TYPE ST_TcMatSimObjectDataAreaInfo :
STRUCT
	pPlcVar: PVOID;
	pModuleProcImg: PVOID;
	nSize: UDINT;
	nDataAreaId: UDINT;
	eDataAreaType: E_TcMatSimDataAreaType;
END_STRUCT
END_TYPE

(* stored: Version 1.1.0.1, ProductVersion 3.1.4020.12
   DUT ST_TcMatSimObjectDataAreaInfo: Id {c0f6f479-068c-4e8d-9041-f68f116a2aef} *)
